(* PLC project CoDeSys External Library Template, WAGO e!COCKPIT e!COCKPIT, author 3S - Smart Software Solutions GmbH *)
(* stored: creationDateTime 2019-10-29T12:37:19.4307338, version 3.5.5.30, modificationDateTime 2019-10-29T12:36:39.3744516, organization 3S - Smart Software Solutions GmbH *)
(* Library project template with all possible element types, docu and a sample project structure *)

(* Autor: Paweł Kąkol, 2018-09-04-PK Prawa majątkowe: Solwena Sp. z o.o., Aktualizacje: 2019-01-28-JC: defrost 2019-02-14-AWy: alarm czujnika temperatury 2019-02-18-AWy: zmiana klas alarmów Opis: enum służy do definicji klas alarmów w fb siłownika (SAB+) HRU0 na budynkach PPP Sopot *)
{attribute 'qualified_only'}
{attribute 'strict'}
TYPE enumPPPSSilownikSABpErrorKlasa : (BrakKomunikacji := enumKlasaAlarmu.AwariaAutomatyki, AlarmOgolny := enumKlasaAlarmu.Ostrzezenie, DetekcjaOtwarciaOkna := enumKlasaAlarmu.Informacyjny, Defrost := enumKlasaAlarmu.Bezpieczenstwa, AlarmCzujnika := enumKlasaAlarmu.AwariaAutomatyki);
END_TYPE
